(* IEC 61131-3 sources: RL_MAR/experiments/comparison/autoplc/results/gpt-4o_20260511_211137/med_74, 1 file *)

(* ---- med_74_1.st ---- *)
FUNCTION_BLOCK TrafficManagementSystem
    VAR_INPUT
        VehicleCount1 : INT; (* Input for vehicle count at intersection 1 *)
        VehicleCount2 : INT; (* Input for vehicle count at intersection 2 *)
        VehicleCount3 : INT; (* Input for vehicle count at intersection 3 *)
        VehicleCount4 : INT; (* Input for vehicle count at intersection 4 *)
    END_VAR
    VAR_OUTPUT
        TrafficLight1 : BOOL; (* Output for traffic light at intersection 1 *)
        TrafficLight2 : BOOL; (* Output for traffic light at intersection 2 *)
        TrafficLight3 : BOOL; (* Output for traffic light at intersection 3 *)
        TrafficLight4 : BOOL; (* Output for traffic light at intersection 4 *)
    END_VAR

    VAR
        (* Internal variables can be declared here if needed *)
    END_VAR

    (* Initialization: Set all traffic lights to a safe state, Red (FALSE) *)
    TrafficLight1 := FALSE;
    TrafficLight2 := FALSE;
    TrafficLight3 := FALSE;
    TrafficLight4 := FALSE;

    (* Continuous Monitoring and Decision Making for Intersection Pair 1 *)
    IF VehicleCount1 > VehicleCount2 THEN
        TrafficLight1 := TRUE;  (* Set TrafficLight1 to Green *)
        TrafficLight2 := FALSE; (* Set TrafficLight2 to Red *)
    ELSE
        TrafficLight1 := FALSE; (* Set TrafficLight1 to Red *)
        TrafficLight2 := TRUE;  (* Set TrafficLight2 to Green *)
    END_IF

    (* Continuous Monitoring and Decision Making for Intersection Pair 2 *)
    IF VehicleCount3 > VehicleCount4 THEN
        TrafficLight3 := TRUE;  (* Set TrafficLight3 to Green *)
        TrafficLight4 := FALSE; (* Set TrafficLight4 to Red *)
    ELSE
        TrafficLight3 := FALSE; (* Set TrafficLight3 to Red *)
        TrafficLight4 := TRUE;  (* Set TrafficLight4 to Green *)
    END_IF

    (* Output Control: The traffic light outputs are updated based on the decision-making logic *)
    (* Persistence and Safety: Ensure the traffic light states persist correctly across task cycles *)
END_FUNCTION_BLOCK
